Yaskawa INFORM job: CVAR_EXAMPLE.JBI

/JOB
//NAME CVAR_EXAMPLE
//POS
///NPOS 9,0,0,0,0,0
///TOOL 0
///POSTYPE PULSE
///PULSE
C00000=0,0,0,0,0,0,0
C00001=-5223,277,-245,333,133,-1223,-1223
C00002=-10446,554,-490,666,266,-2446,-2446
C00003=-15669,831,-735,999,399,-3669,-3669
C00004=-20892,1108,-980,1332,532,-4892,-4892
C00005=-26115,1385,-1225,1665,665,-6115,-6115
C00006=-31338,1662,-1470,1998,798,-7338,-7338
C00007=-36561,1939,-1715,2331,931,-8561,-8561
C00008=-47000,2500,-2200,3000,1200,-11000,-11000
//INST
///DATE 2011/12/21 00:50
///ATTR SC,RW
///GROUP1 RB1
NOP
MOVJ C00000 VJ=25.00
MOVJ C00001 VJ=25.00
MOVJ C00002 VJ=25.00
MOVJ C00003 VJ=25.00
MOVJ C00004 VJ=25.00
MOVJ C00005 VJ=25.00
MOVJ C00006 VJ=25.00
MOVJ C00007 VJ=25.00
MOVJ C00008 VJ=25.00
END
